(* This whole function block is to load cam profiles from a csv file
 * onto the PLC program. This is only temporarily needed to test/learn the cam library.
 * This will not be used when developing the machine, since the cam profiles will be loaded
 * from recipe management.
 *)

FUNCTION_BLOCK FB_CamProfiles
VAR_INPUT
END_VAR
VAR_OUTPUT
END_VAR
VAR
	sFilePath		: STRING;
	
	bReadDone		: BOOL;
	bCreateDone		: BOOL;
END_VAR

METHOD mCreateCamProfiles : BOOL
VAR_INPUT
	Execute			: BOOL;
END_VAR
VAR_IN_OUT
	ALL_CAM			: ARRAY [1..4] OF ARRAY [0..359] OF ARRAY [0..1] OF LREAL;
	ALL_CAM_REF		: ARRAY [1..4] OF MC_CAM_REF;
END_VAR

VAR_INST
	nState			: INT;
	rtStart			: R_TRIG;
	
	nIndex			: INT;
	CamTableSelect	: MC_CamTableSelect;
END_VAR
CASE nState OF
	0:
		rtStart(CLK := Execute);
		IF rtStart.Q THEN
			bCreateDone	:= FALSE;
			nState		:= 5;
		END_IF
	5:
		FOR nIndex := 1 TO 4 DO
			ALL_CAM_REF[nIndex].pArray		:= ADR(ALL_CAM[nIndex]);
			ALL_CAM_REF[nIndex].ArraySize	:= SIZEOF(ALL_CAM[nIndex]);
			ALL_CAM_REF[nIndex].TableType	:= MC_TABLETYPE_EQUIDISTANT;
			ALL_CAM_REF[nIndex].NoOfRows	:= 360;
			ALL_CAM_REF[nIndex].NoOfColumns	:= 2;
		END_FOR
		nIndex 			:= 1;
		nState			:= 10;
	10:
		CamTableSelect(
			Execute		:= TRUE,
			Periodic	:= FALSE,
			CamTableID	:= nIndex,
			CamTable	:= ALL_CAM_REF[nIndex]);
		IF CamTableSelect.Error THEN 
			nState		:= 255;
		ELSIF CamTableSelect.Done AND nIndex < 4 THEN
			CamTableSelect(Execute:=FALSE, CamTable	:= ALL_CAM_REF[nIndex]);
			nIndex		:= nIndex + 1;
		ELSIF CamTableSelect.Done THEN
			CamTableSelect(Execute:=FALSE, CamTable	:= ALL_CAM_REF[nIndex]);
			nState		:= 15;
		END_IF
	15:
		bCreateDone		:= TRUE;
		nState			:= 0;
END_CASE
END_METHOD

METHOD mReadAndStoreSlavePositions : BOOL
VAR_INPUT
	Execute			: BOOL;
END_VAR

VAR_IN_OUT
	ALL_CAM			: ARRAY [1..4] OF ARRAY [0..359] OF ARRAY [0..1] OF LREAL;
END_VAR

VAR_INST
	nState			: INT;
	rtStart			: R_TRIG;
	fbFileOpen		: FB_FileOpen;
	fbFileClose		: FB_FileClose;
	fbFileGets		: FB_FileGets;	// Read 1 csv line function block.
	fileHandle		: UINT;
	
	sReadLine		: STRING;
	
	aPositionStr	: ARRAY [0..360] OF STRING;
	nIndex			: INT;
	nCamFileNumber	: INT := 1;
	lrAbsPosition	: LREAL;
	aTemp			: ARRAY [0..1] OF LREAL;
END_VAR
CASE nState OF
	0:	// IDLE
		rtStart(CLK := Execute);
		IF rtStart.Q THEN
			bReadDone	:= FALSE;
			sReadLine	:= '';
			nIndex		:= 0;
			nState		:= 5;
		END_IF
	5:	// Set file path base Cam profile
		sFilePath		:= 'C:\Users\Administrator\Desktop\Cam_Profiles\8605-005 V2\Slave_';// Path: 	.\
		sFilePath		:= CONCAT(sFilePath, INT_TO_STRING(nCamFileNumber));				//			.\Slave_#
		sFilePath		:= CONCAT(sFilePath, '.csv');										//			.\Slave_#.csv
		nState			:= 10;
	10:	// Open the correspondence CSV file
		fbFileOpen(
			sNetId		:= '10.75.0.183.1.1',
			sPathName	:= sFilePath,
			nMode		:= FOPEN_MODEREAD,
			ePath		:= PATH_GENERIC,
			bExecute	:= TRUE,
			tTimeout	:= DEFAULT_ADS_TIMEOUT);
		nState			:= 15;
	15:	// File open helper state
		fbFileOpen(	bExecute := FALSE, hFile => fileHandle);
		IF NOT fbFileOpen.bBusy AND NOT fbFileOpen.bError THEN
			nState		:= 20;
		ELSIF fbFileOpen.bError THEN
			nState		:= 255;
		END_IF
	20:	// Read 1 line from the openned file, store the line to sReadLine
		fbFileGets(
			sNetId		:= '10.75.0.183.1.1',
			hFile		:= fileHandle,
			bExecute	:= TRUE,
			sLine		=> sReadLine);
		IF NOT fbFileGets.bBusy AND NOT fbFileGets.bError THEN
			// Reset fbFileGets execute flag => remove the read line from memory buffer, so when fbFileGets is called again, the next line is read.
			fbFileGets(bExecute:=FALSE);
			// If not End_Of_File, then append the value to the Position Array and increment the index.
			IF NOT fbFileGets.bEOF THEN
				aPositionStr[nIndex]:= sReadLine;
				nIndex	:= nIndex + 1;
			ELSE
				nIndex	:= 0;
				nState	:= 25;
			END_IF
		ELSIF fbFileGets.bError THEN
				nState	:= 255;
		END_IF
	25:	// 
		FOR nIndex := 0 TO 359 DO
			lrAbsPosition:= STRING_TO_LREAL(aPositionStr[nIndex]);
			aTemp[0]	:= nIndex;
			aTemp[1]	:= lrAbsPosition;
			ALL_CAM[nCamFileNumber][nIndex]:= aTemp;
		END_FOR
		nState			:= 30;
	30:
		nIndex 			:= 0;
		fbFileClose(
			sNetId		:= '10.75.0.183.1.1',
			hFile		:= fileHandle,
			bExecute	:= TRUE);
		nState			:= 35;
	35:
		fbFileClose(bExecute:=FALSE);
		IF NOT fbFileClose.bBusy THEN
			IF NOT fbFileClose.bError THEN
				nState	:= 40;
			ELSE
				nState	:= 255;
			END_IF
		END_IF
	40:
		IF nCamFileNumber < 4 THEN
			nCamFileNumber:= nCamFileNumber + 1;
			nState		:= 5;
		ELSE
			bReadDone	:= TRUE;
			nState		:= 0;
		END_IF
END_CASE
END_METHOD

PROPERTY pCreateDone : BOOL
GET
pCreateDone := bCreateDone;
END_GET
END_PROPERTY

PROPERTY pReadDone : BOOL
GET
pReadDone := bReadDone;
END_GET
END_PROPERTY

END_FUNCTION_BLOCK

(* stored: Version 1.1.0.1, ProductVersion 3.1.4024.15
   POU FB_CamProfiles: Id {bed509b4-f61f-417b-8036-d140481d4bee}, SpecialFunc None
   Method mCreateCamProfiles: Id {2a61a984-6c84-4e75-81a4-8abf3fc2e1ec}
   Method mReadAndStoreSlavePositions: Id {eeef5389-b72d-4ad4-b3db-88221ce8420d}
   Property pCreateDone: Id {5dd09ab0-d193-419d-b396-a1a5cc65b2fd}
   Get Get: Id {21041253-016f-4a13-a545-7be87e7f1e9c}
   Property pReadDone: Id {cd232594-def7-48c2-a74f-2f752c55ce5c}
   Get Get: Id {57296c4b-f6e7-4a4d-9bf5-c6edfaf32da7} *)
